Staubli VAL3: startCycle.pgx

program startCycle(num x_nPoint)
  local string l_sMessage
  local bool l_bOk
  local num l_nSize
  local string l_sButton[2]
begin
  // START
  watch(cycleStatus:nInterfaceToSV==-1,5)
  // get the question message
  call language:message(l_sMessage,214)
  call language:getYesNo(l_sButton)
  // ask the yes_no question
  call use:yes_no(l_sMessage,l_sButton,l_bOk)
  if l_bOk
    // reSTART??
    call trajType:getSizeItem(false,l_nSize)
    if nPoint==l_nSize-1
      x_nPoint=nPoint=0
    endIf
    // compose with 2 element
    cycleStatus:iToSuperV.sType=saveData:sTrajTypeUsing
    cycleStatus:iToSuperV.sData=sTrajName+","+toString("",x_nPoint)
    // send the command to the SuperV
    cycleStatus:nInterfaceToSV=3
    logMsg("[KERNEL] INTERFACE:Simulation of the item: "+saveData:sTrajTypeUsing+" "+sTrajName)
    // wait the command has been receive
    watch(cycleStatus:nInterfaceToSV==-1,5)
  endIf
end
